INTERFACE I_LoggerFactory EXTENDS I_Logger

{attribute 'OPC.UA.DA.Property' := '1'}
{attribute 'monitoring' := 'call'}
PROPERTY PUBLIC P_Events : reference to ARRAY [0..Parameters.nEvents] OF ST_Event
GET
END_GET
END_PROPERTY

{attribute 'OPC.UA.DA.Property' := '1'}
{attribute 'monitoring' := 'call'}
PROPERTY PUBLIC P_Length : DINT
GET
END_GET
END_PROPERTY

END_INTERFACE

(* stored: Version 1.1.0.1
   Itf I_LoggerFactory: Id {1075ed47-adad-0375-2b61-454fd2394881}
   Property P_Events: Id {82907ad1-f2c2-0828-09af-9aabebd52ddb}
   Get Get: Id {64b0b94a-59f5-0f06-145c-b91fed7ca0e8}
   Property P_Length: Id {db5a6d16-914e-04ec-2a29-d57635ae33cc}
   Get Get: Id {0d198b76-c71f-00b8-1fcc-6cc00a90a1b4} *)
